// TwinCAT 3 PLC project Examples
// ProgramVersion: 3.1.4024.0
// libraries:
//   Tc2_Standard, * (Beckhoff Automation GmbH)
//   Tc2_System, * (Beckhoff Automation GmbH)
//   Tc3_Module, * (Beckhoff Automation GmbH)
//   Tc3_UnitTest, * (Zerlauth)
// project tree:
//   GVLs/ FB_Target.TcPOU, FB_UnitTestTarget01.TcPOU, FB_UnitTestTarget02.TcPOU, GVL.TcGVL
//   POUs/ MAIN.TcPOU
// (motion and I/O tree: see PLC project tc3_unittest)
// real-time tasks:
//   TASK PlcTask: cycle T#10ms, priority 20, ADS port 350

// ---- GVLs/GVL.TcGVL
	{attribute 'analysis' := '-27'}
VAR_GLOBAL

	fbTestsuites:			FB_Testsuites;				// Testsuites
END_VAR

// ---- GVLs/FB_Target.TcPOU
FUNCTION_BLOCK FB_Target
VAR_INPUT
END_VAR
VAR_OUTPUT
END_VAR
VAR
END_VAR

END_FUNCTION_BLOCK

// ---- GVLs/FB_UnitTestTarget01.TcPOU
FUNCTION_BLOCK FB_UnitTestTarget01 EXTENDS FB_Target
VAR_INPUT
END_VAR
VAR_OUTPUT
END_VAR
VAR
	fbTestsuite:			FB_Testsuite;				// Testsuite
	sValue:					STRING;
END_VAR

SUPER^();

fbTestsuite();


CASE fbTestsuite.P_Testcase OF
	E_Testcase.Init:
		sValue:= 'Test';

	E_Testcase.Start:
		// First test case
		fbTestsuite.P_Assert.M_Equals_STRING('Test', sValue, 'Check string value "Test"');
		fbTestsuite.M_Testcase('FB_Target', T#1S, '', '', 1);
		
	// secound test case
	1:
		fbTestsuite.P_Assert.M_IsTRUE('Test2' <> sValue, 'Check string value "Test2"');
		fbTestsuite.M_Testcase('FB_Target', T#1S, '', '', E_Testcase.Done);
		
	E_Testcase.Done:
		
END_CASE

METHOD FB_init : BOOL
VAR_INPUT
	bInitRetains : BOOL; // if TRUE, the retain variables are initialized (warm start / cold start)
	bInCopyCode : BOOL;  // if TRUE, the instance afterwards gets moved into the copy code (online change)
END_VAR
//// Add Testsuite to Testsuites
fbTestsuites.M_Add(fbTestsuite);
fbTestsuite.P_File:= 'FB_Target';
END_METHOD

END_FUNCTION_BLOCK

// ---- GVLs/FB_UnitTestTarget02.TcPOU
FUNCTION_BLOCK FB_UnitTestTarget02 EXTENDS FB_Target
VAR_INPUT
END_VAR
VAR_OUTPUT
END_VAR
VAR
	fbTestsuite:			FB_Testsuite;				// Testsuite
	sValue:					STRING;
END_VAR

SUPER^();

fbTestsuite();


CASE fbTestsuite.P_Testcase OF
	E_Testcase.Init:
		sValue:= 'Test';

	E_Testcase.Start:
		// First test case
		fbTestsuite.P_Assert.M_Equals_STRING('Test', sValue, 'Check string value "Test"');
		fbTestsuite.M_Testcase('FB_Target', T#1S, '', '', 1);
		
	// secound test case
	1:
		fbTestsuite.P_Assert.M_IsTRUE('Test2' <> sValue, 'Check string value "Test2"');
		fbTestsuite.M_Testcase('FB_Target', T#1S, '', '', E_Testcase.Done);
		
	E_Testcase.Done:
		
END_CASE

METHOD FB_init : BOOL
VAR_INPUT
	bInitRetains : BOOL; // if TRUE, the retain variables are initialized (warm start / cold start)
	bInCopyCode : BOOL;  // if TRUE, the instance afterwards gets moved into the copy code (online change)
END_VAR
//// Add Testsuite to Testsuites
fbTestsuites.M_Add(fbTestsuite);
fbTestsuite.P_File:= 'FB_Target';
END_METHOD

END_FUNCTION_BLOCK

// ---- POUs/MAIN.TcPOU
PROGRAM MAIN
VAR
	bExecute:					BOOL;
	fbFunctionBlock01:		FB_UnitTestTarget01;
	fbFunctionBlock02:		FB_UnitTestTarget02;
END_VAR

// Run
fbTestsuites();

IF bExecute THEN
	bExecute:= NOT fbTestsuites.M_Request(E_Base.Execute);
END_IF

fbFunctionBlock01();
fbFunctionBlock02();

END_PROGRAM
